PROGRAM MAIN
VAR
END_VAR

PB_TestRunner();

END_PROGRAM

(* stored: Version 1.1.0.1, ProductVersion 3.1.4024.4
   POU MAIN: Id {98813dcb-669b-4314-a691-09db98998046}, SpecialFunc None *)
